// TwinCAT 3 PLC project NinjaTest
// ProgramVersion: 3.1.4026.12
// libraries:
//   Tc2_Standard, * (Beckhoff Automation GmbH)
//   Tc2_System, * (Beckhoff Automation GmbH)
//   Tc2_Utilities, * (Beckhoff Automation GmbH)
// project tree:
//   DUTs/ E_Example.TcDUT
//   GVLs/ GVL.TcGVL
//   Implicit Checks/ CheckRangeSigned.TcPOU, CheckRangeUnsigned.TcPOU
//   / PlcTask.TcTTO, PRG_Alt.TcPOU
//   POUs/Examples/Factory/Devices/ FB_AbstractDevice.TcPOU, FB_PressureTransducer.TcPOU, FB_TemperatureTransducer.TcPOU, FB_Solonoid.TcPOU, I_Device.TcIO
//   POUs/Examples/Factory/Devices/Types/Alias/ A_Devices.TcDUT
//   POUs/Examples/Factory/Devices/Types/Enumerations/ E_DeviceTypes.TcDUT
//   POUs/Examples/Factory/ FB_FactoryExample.TcPOU, F_DeviceFactory.TcPOU
//   POUs/Examples/ FB_ArrayExample.TcPOU, FB_DefaultInputExample.TcPOU, FB_DynamicMemoryExample.TcPOU, FB_JumpAndReturnExample.TcPOU, FB_OneShotExample.TcPOU, FB_SelectOperatorExample.TcPOU, FB_SubRangeExample.TcPOU, FB_ToTypeExample.TcPOU, FB_EnumAndCaseExample.TcPOU, FB_ForWhileRepeatExample.TcPOU
//   POUs/Examples/Function Block/ FB_FunctionBlockExample.TcPOU
//   POUs/Examples/Function Block/Helpers/ FB_Abstract.TcPOU, FB_AbstractChild.TcPOU, FB_Final.TcPOU, FB_FinalChild.TcPOU, FB_InstanceVariables.TcPOU
//   POUs/Helpers/ FB_Test.TcPOU, I_Test.TcIO
//   POUs/ MAIN.TcPOU
// real-time tasks:
//   TASK PlcTask: cycle T#10ms, priority 20, ADS port 350

CONFIGURATION NinjaTest
    RESOURCE PLC ON TwinCAT3
        TASK PlcTask(INTERVAL := T#10ms, PRIORITY := 20);
        PROGRAM MAIN WITH PlcTask : MAIN;
        PROGRAM PRG_Alt WITH PlcTask : PRG_Alt;
    END_RESOURCE
END_CONFIGURATION

// ---- DUTs/E_Example.TcDUT
{attribute 'qualified_only'}
{attribute 'strict'}
{attribute 'to_string'}
TYPE E_Example :
(
	red := -1,
	blue,
	green
) SINT := blue; //Definfes this as a SINT with a default value of blue
END_TYPE

// ---- POUs/Examples/Factory/Devices/Types/Alias/A_Devices.TcDUT
TYPE A_Devices : INT(1..3); END_TYPE

// ---- POUs/Examples/Factory/Devices/Types/Enumerations/E_DeviceTypes.TcDUT
{attribute 'qualified_only'}
{attribute 'strict'}
{attribute 'to_string'}
TYPE E_DeviceTypes :
(
	PressureTransducer := 0,
	TemperatureTransducer,
	Solonoid
);
END_TYPE

// ---- GVLs/GVL.TcGVL
{attribute 'qualified_only'}
VAR_GLOBAL CONSTANT
	INDEX_MIN : INT := 1;
	INDEX_MAX : INT := 10;
END_VAR

// ---- POUs/Examples/Factory/Devices/I_Device.TcIO
INTERFACE I_Device

PROPERTY name : STRING
GET
END_GET
SET
END_SET
END_PROPERTY

END_INTERFACE

// ---- POUs/Helpers/I_Test.TcIO
INTERFACE I_Test

METHOD M_Cyclic
VAR_INPUT
END_VAR
END_METHOD

END_INTERFACE

// ---- POUs/MAIN.TcPOU
PROGRAM MAIN

VAR
	// Examples
	totype : FB_ToTypeExample;
	defaultInput : FB_DefaultInputExample;
	subRangeExample : FB_SubRangeExample;
	selectOperator : FB_SelectOperatorExample;
	arraryExample : FB_ArrayExample;
	enumAndCaseExample : FB_EnumAndCaseExample;
	jumpAndReturnExample : FB_JumpAndReturnExample;
	forWhilERepeatExample : FB_ForWhileRepeatExample;
	oneShotExample : FB_OneShotExample;
	functionBlockExample : FB_FunctionBlockExample;
	dynamicMemory : FB_DynamicMemoryExample;
	factoryExample : FB_FactoryExample;
END_VAR

// TO_(Type)
totype();

// As of 4026 do not need to specify inputs with default values
defaultInput();

// Subrange datatype, can see been usful for range
subRangeExample();

// LIMIT and SEL
selectOperator();

// Array with variable length
arraryExample();

// Enum and Case Statement
enumAndCaseExample();

// Jump & Return
jumpAndReturnExample();

// For, While and Repeat
forWhilERepeatExample();

// Example of how to do a one shot
oneShotExample();

// Function Block
functionBlockExample();

// Reference during FB_Ini and dynamic creation of FB, moved to FB so we can use FB_Exit to delete the mmemory
dynamicMemory();

// Factory
factoryExample();

// factoryExample.PT01.name // example of a PT call

END_PROGRAM

// ---- POUs/Examples/FB_ToTypeExample.TcPOU
FUNCTION_BLOCK FB_ToTypeExample

VAR
	// To_type
	test1 : UDINT := 5;
	result1 : SINT;

	test2 : BOOL := TRUE;	
	result2a : STRING;
	result2b : INT;
END_VAR

// Note yo udo not need to specif the from conition in a explicit conversion i.e. UDINT_TO_INT(5) can be wrriten as TO_INT(5).
// Form that the conversion takes depends on what you are convering from i.e. TO_STRING(TRUE) = "TRUE" where as TO_INT(TRUE) = 1.

// TO_(Type)
result1 := TO_SINT(test1); // Change to > 255 and see what reult 1 behaves

result2a := TO_STRING(test2);
result2b := TO_INT(test2);

END_FUNCTION_BLOCK

// ---- POUs/Examples/FB_DefaultInputExample.TcPOU
FUNCTION_BLOCK FB_DefaultInputExample

VAR	
	// Default values of VAR_INPUT
	test, result1, result2 : INT;
END_VAR

// Fully defined input
result1 := M_Addition(input1 := test, input2 := 20);

// On required field declared, input2 has a default value of 25
result2 := M_Addition(input1 := test);

METHOD M_Addition :INT

VAR_INPUT
	input1 : INT;
	input2 : INT := 25;
END_VAR
M_Addition := input1 + input2;
END_METHOD

END_FUNCTION_BLOCK

// ---- POUs/Examples/FB_SubRangeExample.TcPOU
FUNCTION_BLOCK FB_SubRangeExample

VAR
	// Sub range
	test1 : INT(1..2);

	test2 : INT(GVL.INDEX_MIN..GVL.INDEX_MAX);
	test3 : INT := 15;
END_VAR

// Could be useful for setting up index for for loops

// Can be used with Alias to create parameters i.e. we could have a ALIAS of mARaw which contains UINT(4000...20000) this way we know we will only get the mA and not outside ranges

test1 := 2;
// test1 := 4;// Will result in compile error as it is out of range

test2 := test3; // Without implicit checks it will take the value of test3, with implicit checks it will take the max range.

END_FUNCTION_BLOCK

// ---- POUs/Examples/FB_SelectOperatorExample.TcPOU
FUNCTION_BLOCK FB_SelectOperatorExample

VAR
	test1, result1, result2, lowerLimit, upperLimit : DINT;
	test2 : BOOL;
END_VAR

result1 := LIMIT(lowerLimit, test1 ,upperLimit);

result2 := SEL(test2, 1, 2);

END_FUNCTION_BLOCK

// ---- POUs/Examples/FB_ArrayExample.TcPOU
FUNCTION_BLOCK FB_ArrayExample

VAR
	test1 : ARRAY[GVL.INDEX_MIN..5] OF INT := [5,8, 9, 6, 7];
	test2 : ARRAY[1..10] OF INT := [10(8)]; // Will all be initalised with 8
	answer1, answer2 : DINT;
END_VAR

answer1 := M_SumArray(test1);
answer2 := M_SumArray(test2);

METHOD M_SumArray : DINT

VAR_IN_OUT
	data : ARRAY[*] OF INT;
END_VAR

VAR
	i, sum : DINT;
END_VAR
RETURN ( LEN2(DATA) < 1 );

FOR i := LOWER_BOUND(data, 1) TO UPPER_BOUND(data, 1) DO
	sum := sum + data[i];
END_FOR

M_SumArray := sum;
END_METHOD

END_FUNCTION_BLOCK

// ---- POUs/Examples/FB_EnumAndCaseExample.TcPOU
FUNCTION_BLOCK FB_EnumAndCaseExample

VAR
	//Enum and case
	test1 : E_Example;
	result1a : STRING;
	result1b : STRING;
	
	test2 : INT;
	result2 : STRING;
END_VAR

// Enum and case
CASE test1 OF
	E_Example.blue :
		result1a := 'Blue';
	E_Example.green :
		result1a := 'Green';
	E_Example.red :
		result1a := 'Red';
	ELSE
		result1a := '';
END_CASE
result1b := TO_STRING(test1);

CASE test2 OF
	1       : result2 := '1';
	2,3,4,5 : result2 := 'Between 2 and 5';
	6..20   : result2 := 'Between 6 and 20';
ELSE     
	result2 := 'Greater than 20';
END_CASE

END_FUNCTION_BLOCK

// ---- POUs/Examples/FB_JumpAndReturnExample.TcPOU
FUNCTION_BLOCK FB_JumpAndReturnExample

VAR
	jump1, jump2, return1, return2: BOOL;
	pointerValid, referenceValid : BOOL := TRUE;
	ptr : POINTER TO STRING;
	ref : REFERENCE TO STRING;
	msg : STRING := 'This is a msg';
	jmpResult : STRING;
END_VAR

IF pointerValid THEN
	ptr := ADR(msg); 
ELSE
	ptr := 0;// Manually zero out the pointer
END_IF

IF referenceValid THEN
	ref REF= msg;
ELSE
	ref REF= 0; // Invlaid type for this reference
END_IF
	
M_TestMethod(jump1 := jump1, jump2 := jump2, return1 := return1, return2 := return2, ptr := ptr, ref := ref, result => jmpResult);

METHOD M_TestMethod

VAR_INPUT
	jump1, jump2 : BOOL;
	return1, return2 : BOOL;
	ref : REFERENCE TO STRING;
	ptr : POINTER TO STRING;
END_VAR

VAR_OUTPUT
	result : STRING;
END_VAR

// This can be useful if you want a override which skips some of the code, 
// i.e. you have code which does a action then monitors the result, you may want a override which skips the control if disabled but still monitors
// Return via a if statement
IF return1 THEN
	result := 'I returned early due to return1';
	RETURN;
END_IF

// Conditional Returns
result := 'I returned early due to return2';
RETURN ( return2 );

result := 'I returned early due to a invalid reference';
RETURN ( NOT __ISVALIDREF(ref) );

result := 'I returned early due to a invalid pointer';
RETURN ( ptr = 0 );

// Jump via a if statement
IF jump1 THEN
	JMP j1;
END_IF

// Jump via a condition jump
JMP ( jump2 ) j2;

// Default Answer
result := 'I have not jumped';
RETURN;

j1: result := 'I have jumped using jump 1';	
RETURN;

j2: result := 'I have jumped using jump 2';	
RETURN;
END_METHOD

END_FUNCTION_BLOCK

// ---- POUs/Examples/FB_ForWhileRepeatExample.TcPOU
FUNCTION_BLOCK FB_ForWhileRepeatExample 

VAR
	test : INT := 2;
	result1, result2, result3 : DINT;
	healthy2, healthy3 : BOOL;
END_VAR

// For
M_For(sum => result1);

M_ForAdvanced();

// While
healthy2 := M_While(condition := test, count => result2);

// Repeat
healthy3 := M_Repeat(condition := test, count => result3);

METHOD M_For : BOOL

VAR
	test : ARRAY[1..10] OF INT :=  [10(2)];
	i : INT;
END_VAR

VAR_OUTPUT
	sum : DINT;
END_VAR
FOR i := 1 TO 10 BY 1 DO
	sum := sum + test[i];
END_FOR
END_METHOD

METHOD M_ForAdvanced : BOOL

VAR
	i : INT;
	sum : DINT;
	
	test : REFERENCE TO INT REF= 0;
END_VAR
FOR i := 1 TO 10 DO
	IF i > 5 THEN
		test REF= i;	
	END_IF

// Will crash as we try to use a invalid REFERENCE	
//	IF NOT (__ISVALIDREF(test) AND test  > 7 ) THEN		
//		CONTINUE;
//	END_IF

// Will not crash as we test the reference before we use it
	IF NOT (__ISVALIDREF(test) AND_THEN test  > 7 ) THEN		
		CONTINUE;
	END_IF

	sum := sum + 1;	
END_FOR
END_METHOD

METHOD M_Repeat : BOOL
VAR_INPUT
	condition : INT;
END_VAR

VAR_OUTPUT
	count : DINT;
END_VAR

VAR
	test : ARRAY[1..10] OF INT := [1,2,3,4,5,6,7,8,9,10];
	i : INT := 1;;
END_VAR

// Similar to the while loop but will always do one cycle as it tests the condition til the end
M_Repeat := FALSE;
RETURN ( condition < 1 OR condition > 10 );

REPEAT
	count := count + test[i];
	IF i > 10 THEN
		EXIT;
	END_IF
	i:= i + 1;
UNTIL
	test[i] = condition
END_REPEAT

M_Repeat := TRUE;
END_METHOD

METHOD M_While : BOOL

VAR_INPUT
	condition : INT;
END_VAR

VAR_OUTPUT
	count : DINT;
END_VAR

VAR
	test : ARRAY[1..10] OF INT := [1,2,3,4,5,6,7,8,9,10];
	i : INT := 1;;
END_VAR

// Use while with caudition as it can lead to infinite loop
M_While :=FALSE;
RETURN ( condition < 1 OR condition > 10 );

WHILE ( test[i] <> condition ) DO
	count := count + test[i];
	IF i > 10 THEN
		EXIT;
	END_IF
	i:= i + 1;
END_WHILE

M_While := TRUE;
END_METHOD

END_FUNCTION_BLOCK

// ---- POUs/Examples/FB_OneShotExample.TcPOU
FUNCTION_BLOCK FB_OneShotExample
VAR
	execute : BOOL;
END_VAR

M_OneShot(execute);

METHOD M_OneShot

VAR_INPUT
	_execute : BOOL;
END_VAR

VAR_INST
	execTrig : R_Trig;
END_VAR
execTrig(CLK := _execute);
RETURN (NOT execTrig.Q);

// Do code here, will only be called for each time _execute does from low to high
END_METHOD

END_FUNCTION_BLOCK

// ---- POUs/Examples/Function Block/FB_FunctionBlockExample.TcPOU
FUNCTION_BLOCK FB_FunctionBlockExample

VAR
//	abstractExaple : FB_Abstract;  				// Compile error as this FB is abract class
	abstractChildExaple : FB_AbstractChild;
	finalExaple : FB_Final;
	finalChildExaple : FB_FinalChild;
	
	instantVariables : FB_InstanceVariables;
END_VAR

// abstractExaple();

abstractChildExaple();

finalExaple();

finalChildExaple();

instantVariables();

END_FUNCTION_BLOCK

// ---- POUs/Examples/Function Block/Helpers/FB_AbstractChild.TcPOU
FUNCTION_BLOCK FB_AbstractChild EXTENDS FB_Abstract
VAR_INPUT
END_VAR
VAR_OUTPUT
END_VAR
VAR
END_VAR

{warning 'Add method implementation '} //  Auto generated due to child class being Abstract
METHOD PROTECTED M_Init : BOOL
END_METHOD

END_FUNCTION_BLOCK

// ---- POUs/Examples/Function Block/Helpers/FB_Abstract.TcPOU
FUNCTION_BLOCK ABSTRACT FB_Abstract


// This Function Block can't be instaniated but has to be extended.

METHOD PROTECTED M_Cycle : BOOL
VAR_INPUT
END_VAR

// This Method does not have to be incorporated into child class
END_METHOD

METHOD PROTECTED ABSTRACT M_Init : BOOL
VAR_INPUT
END_VAR


// This Method has to be incorporated into child class
END_METHOD

END_FUNCTION_BLOCK

// ---- POUs/Examples/Function Block/Helpers/FB_Final.TcPOU
FUNCTION_BLOCK FINAL FB_Final


// This Function Block Can't be extended

END_FUNCTION_BLOCK

// ---- POUs/Examples/Function Block/Helpers/FB_FinalChild.TcPOU

// This will fail as FB_Final is Final and can't be extended
//FUNCTION_BLOCK FB_FinalChild EXTENDS FB_Final

// This will fail as FB_Final is Final and can't be extended
 FUNCTION_BLOCK FB_FinalChild

END_FUNCTION_BLOCK

// ---- POUs/Examples/Function Block/Helpers/FB_InstanceVariables.TcPOU
FUNCTION_BLOCK FB_InstanceVariables

VAR
	test1, test2 : INT;
END_VAR

// This stays the same as the variable which we increment is reset on each call as its a var
test1 := M_AddLocal();

// This increases as the variable which we increment is added to the FB memory and is keep each cycle as its a var_inst
test2 := M_AddInst();

METHOD M_AddInst : INT

VAR_INST
	current : INT;
END_VAR
current := current + 1;

M_AddInst := current;
END_METHOD

METHOD M_AddLocal : INT

VAR
	current : INT;
END_VAR
current := current + 1;

M_AddLocal := current;
END_METHOD

END_FUNCTION_BLOCK

// ---- POUs/Examples/FB_DynamicMemoryExample.TcPOU
FUNCTION_BLOCK FB_DynamicMemoryExample

VAR
	initalize : BOOL;
		
	test : POINTER TO FB_Test;
	test2 : REFERENCE TO FB_Test;
	test3 : I_Test;
	
	test4 : FB_Test(processRef := PRG_Alt.test) := (name := 'test04');
	
	intialised : BOOL;
	initTrig : R_TRIG;
END_VAR

// This is a example of how you can use JMP and return, should create a init and cyclic logic methods and use the initialised to call the different code. 
// But could be useful for functions which do not support methods, or simple overrides [i.e. HMI or enable overrides]

initTrig(CLK := initalize);

JMP ( NOT intialised ) init;
JMP ( intialised ) cycle;

init: // Initalise
RETURN ( NOT initTrig.Q ); // Do nothing unless told to

test := __NEW( FB_Test(processRef := PRG_Alt.test) );
test^.name :='test';
IF test <> 0 THEN
	test2 REF= test^;
	test3 := test^;
END_IF
intialised := TRUE;	
RETURN;

cycle: // After Initalise
RETURN ( test = 0 );
test^(); // Deferance pointer and call directly [use only as needed]

RETURN ( NOT __ISVALIDREF(test2) );
test2();  // Call via the reference [better option]

// Continue code ...
test3.M_Cyclic(); // Call via a interfadce [prefered option, no check required]

test4();
RETURN;

//FB_Exit must be implemented explicitly. If there is an implementation, then the
//method is called before the controller removes the code of the function block instance
//(implicit call). The return value is not evaluated.
METHOD FB_Exit: BOOL
VAR_INPUT
    bInCopyCode: BOOL;  // TRUE: the exit method is called in order to leave the instance which will be copied afterwards (online change).  
END_VAR
__delete(test);
END_METHOD

PROPERTY pTest : REFERENCE TO FB_Test;
GET
IF test <> 0 THEN
	pTest REF= test^;
END_IF
END_GET
END_PROPERTY

END_FUNCTION_BLOCK

// ---- POUs/Helpers/FB_Test.TcPOU
{attribute 'enable_dynamic_creation'}
FUNCTION_BLOCK FB_Test IMPLEMENTS I_Test

VAR
	_processRef : REFERENCE TO REAL;
	_name : STRING;
END_VAR

//FB_Init is always available implicitly and it is used primarily for initialization.
//The return value is not evaluated. For a specific influence, you can also declare the
//methods explicitly and provide additional code there with the standard initialization
//code. You can evaluate the return value.
METHOD FB_Init: BOOL
VAR_INPUT
    bInitRetains: BOOL; // TRUE: the retain variables are initialized (reset warm / reset cold)
    bInCopyCode: BOOL;  // TRUE: the instance will be copied to the copy code afterward (online change)   
	processRef : REFERENCE TO REAL;
END_VAR
_processRef REF= processRef;
END_METHOD

METHOD M_Cyclic
END_METHOD

PROPERTY name : STRING
GET
name : _name;
END_GET
SET
_name := name;
END_SET
END_PROPERTY

END_FUNCTION_BLOCK

// ---- PRG_Alt.TcPOU
PROGRAM PRG_Alt
VAR
	test : REAL;
	PT : REAL := 50.5;
	TT : REAL := 11.5;
	SV : BOOL;
END_VAR

END_PROGRAM

// ---- POUs/Examples/Factory/FB_FactoryExample.TcPOU
{attribute 'call_after_init'}
FUNCTION_BLOCK FB_FactoryExample

VAR
	Initialized : BOOL;

	testI : ARRAY[1..NO_OF_DEVICES] OF I_Device;

	{attribute 'hide'} 
	testPtr : ARRAY[1..NO_OF_DEVICES] OF POINTER TO FB_AbstractDevice;
END_VAR

VAR CONSTANT
	NO_OF_DEVICES : A_Devices := 3;
END_VAR

// I would imagine one fo each function blcok for each type of devices similar to HyQube V3 , were we have a interface for each type.

//FB_Exit must be implemented explicitly. If there is an implementation, then the
//method is called before the controller removes the code of the function block instance
//(implicit call). The return value is not evaluated.
METHOD FB_Exit: BOOL
VAR_INPUT
    bInCopyCode: BOOL;  // TRUE: the exit method is called in order to leave the instance which will be copied afterwards (online change).  
END_VAR

VAR
	i : A_Devices;
END_VAR
// Add in check for to ensure it is dynamic type before deletion.
FOR i := 1 TO NO_OF_DEVICES DO
	IF testPtr[i] <> 0 THEN
		__DELETE(testPtr[i]);	
	END_IF
END_FOR
END_METHOD

{attribute 'call_after_init'}
METHOD M_Init : BOOL

VAR
	i : int;
END_VAR
// Dynamically Create blocks and assign 
i := 1;
IF testPtr[i] = 0 THEN
	testPtr[i] := F_DeviceFactory(device := E_DeviceTypes.PressureTransducer, realRef := PRG_Alt.PT);	
	testI[i] := testPtr[i]^;
	testI[i].name := 'PT-01';	
END_IF

i := 2;
IF testPtr[i] = 0 THEN
	testPtr[i] := F_DeviceFactory(device := E_DeviceTypes.TemperatureTransducer, realRef := PRG_Alt.TT);
	testI[i] := testPtr[i]^;
	testI[i].name := 'TT-01';
END_IF

i := 3;
IF testPtr[i] = 0 THEN
	testPtr[i ] := F_DeviceFactory(device := E_DeviceTypes.Solonoid, boolRef := PRG_Alt.SV);
	testI[i] := testPtr[i]^;
	testI[i].name := 'SV-01';
END_IF

Initialized := TRUE;
END_METHOD

PROPERTY PT01 : I_Device
GET
PT01 := testI[1];
END_GET
END_PROPERTY

PROPERTY SV01 : I_Device
GET
SV01 := testI[3];
END_GET
END_PROPERTY

PROPERTY TT01 : I_Device
GET
TT01 := testI[2];
END_GET
END_PROPERTY

END_FUNCTION_BLOCK

// ---- POUs/Examples/Factory/Devices/FB_AbstractDevice.TcPOU
FUNCTION_BLOCK ABSTRACT FB_AbstractDevice IMPLEMENTS I_Device

VAR
	_name : STRING;
END_VAR

PROPERTY name : STRING
GET
name : _name;
END_GET
SET
_name := name;
END_SET
END_PROPERTY

END_FUNCTION_BLOCK

// ---- POUs/Examples/Factory/F_DeviceFactory.TcPOU
FUNCTION F_DeviceFactory : POINTER TO FB_AbstractDevice

VAR_INPUT
	device : E_DeviceTypes;
	boolRef : REFERENCE TO BOOL REF= 0;
	intRef : REFERENCE TO INT REF= 0;
	realRef : REFERENCE TO REAL REF= 0;
END_VAR

VAR
	pressureTransducer : POINTER TO FB_PressureTransducer;
	temperatureeTransducer : POINTER TO FB_TemperatureTransducer;
	solonoid : POINTER TO FB_Solonoid;
END_VAR

CASE device OF
	E_DeviceTypes.PressureTransducer :
		RETURN ( NOT __ISVALIDREF(realRef) );
		pressureTransducer  := __NEW( FB_PressureTransducer(processRef := realRef) );
		F_DeviceFactory := pressureTransducer;
	E_DeviceTypes.TemperatureTransducer :
		RETURN ( NOT __ISVALIDREF(realRef) );
		temperatureeTransducer  := __NEW( FB_TemperatureTransducer(processRef := realRef) );
		F_DeviceFactory := temperatureeTransducer;
	E_DeviceTypes.Solonoid :
		RETURN ( NOT __ISVALIDREF(boolRef) );
		solonoid  := __NEW( FB_Solonoid(output  := boolRef) );
		F_DeviceFactory := solonoid;
END_CASE

END_FUNCTION

// ---- POUs/Examples/Factory/Devices/FB_PressureTransducer.TcPOU
{attribute 'call_after_init'}
{attribute 'enable_dynamic_creation'}
FUNCTION_BLOCK FINAL FB_PressureTransducer EXTENDS FB_AbstractDevice IMPLEMENTS I_Device

VAR
	_processRef : REFERENCE TO REAL;
END_VAR

//FB_Init is always available implicitly and it is used primarily for initialization.
//The return value is not evaluated. For a specific influence, you can also declare the
//methods explicitly and provide additional code there with the standard initialization
//code. You can evaluate the return value.
METHOD FB_Init: BOOL
VAR_INPUT
    bInitRetains: BOOL; // TRUE: the retain variables are initialized (reset warm / reset cold)
    bInCopyCode: BOOL;  // TRUE: the instance will be copied to the copy code afterward (online change)   
	processRef : REFERENCE TO REAL;
END_VAR
_processRef REF= processRef;
END_METHOD

END_FUNCTION_BLOCK

// ---- POUs/Examples/Factory/Devices/FB_TemperatureTransducer.TcPOU
{attribute 'call_after_init'}
{attribute 'enable_dynamic_creation'}
FUNCTION_BLOCK FINAL FB_TemperatureTransducer EXTENDS FB_AbstractDevice IMPLEMENTS I_Device

VAR
	_processRef : REFERENCE TO REAL;
END_VAR

//FB_Init is always available implicitly and it is used primarily for initialization.
//The return value is not evaluated. For a specific influence, you can also declare the
//methods explicitly and provide additional code there with the standard initialization
//code. You can evaluate the return value.
METHOD FB_Init: BOOL
VAR_INPUT
    bInitRetains: BOOL; // TRUE: the retain variables are initialized (reset warm / reset cold)
    bInCopyCode: BOOL;  // TRUE: the instance will be copied to the copy code afterward (online change)   
	processRef : REFERENCE TO REAL;
END_VAR
_processRef REF= processRef;
END_METHOD

END_FUNCTION_BLOCK

// ---- POUs/Examples/Factory/Devices/FB_Solonoid.TcPOU
{attribute 'call_after_init'}
{attribute 'enable_dynamic_creation'}
FUNCTION_BLOCK FINAL FB_Solonoid EXTENDS FB_AbstractDevice IMPLEMENTS I_Device

VAR
	_output : REFERENCE TO BOOL;
END_VAR

//FB_Init is always available implicitly and it is used primarily for initialization.
//The return value is not evaluated. For a specific influence, you can also declare the
//methods explicitly and provide additional code there with the standard initialization
//code. You can evaluate the return value.
METHOD FB_Init: BOOL
VAR_INPUT
    bInitRetains: BOOL; // TRUE: the retain variables are initialized (reset warm / reset cold)
    bInCopyCode: BOOL;  // TRUE: the instance will be copied to the copy code afterward (online change)   
	output : REFERENCE TO BOOL;
END_VAR
_output REF= output;
END_METHOD

END_FUNCTION_BLOCK

// ---- Implicit Checks/CheckRangeSigned.TcPOU
// Implicitly generated code : DO NOT EDIT
FUNCTION CheckRangeSigned : DINT
VAR_INPUT
	value, lower, upper: DINT;
END_VAR

// Implicitly generated code: Only an implementation suggestion
{noflow}
IF (value < lower) THEN
	CheckRangeSigned := lower;
ELSIF(value > upper) THEN
	CheckRangeSigned := upper;
ELSE
	CheckRangeSigned := value;
END_IF

END_FUNCTION

// ---- Implicit Checks/CheckRangeUnsigned.TcPOU
// Implicitly generated code : DO NOT EDIT
FUNCTION CheckRangeUnsigned : UDINT
VAR_INPUT
	value, lower, upper: UDINT;
END_VAR

// Implicitly generated code: Only an implementation suggestion
{noflow}
IF (value < lower) THEN
	CheckRangeUnsigned := lower;
ELSIF(value > upper) THEN
	CheckRangeUnsigned := upper;
ELSE
	CheckRangeUnsigned := value;
END_IF

END_FUNCTION
